Universal Robots PolyScope program: default.urp

Program default (installation=default directory=/ursim/programs createdIn=5.23.0 lastSavedIn=5.23.0 robotSerialNumber=20195599999)
Calibrated DH parameters: a=[0, -0.425, -0.3922, 0, 0, 0]; d=[0.1625, 0, 0, 0.1333, 0.0997, 0.0996]; alpha=[1.570796, 0, 0, 1.570796, -1.570796, 0]; deltaTheta=[0, 0, 0, 0, 0, 0]
InitVariablesNode
Robot Program (runOnlyOnce=false)
  Placeholder
Thread Thread_1 (runOnlyOnce=false)
  Loop Forever
    Script: set_digital_in(1, True )
    Wait Sleep waitTime=0.5
    Script: set_digital_in(1, False )
    Wait Sleep waitTime=0.5
